KUKA KRL data list: $config.dat

&ACCESS RV
&PARAM DISKPATH = SYSTEM
&REL 3
DEFDAT $CONFIG
;FOLD BASISTECH GLOBALS
;==================================
; Default parameters for movement
; These values shouldn't be changed
;==================================

;----------------------------------
; general MOVEMENT - parameters:
;----------------------------------

INT DEF_OV_PRO=100
INT DEF_ADVANCE=3

; PTP - MOVEMENTS
;----------------------------------
INT DEF_VEL_PTP=100
INT DEF_ACC_PTP=50

; CP - MOVEMENTS
;----------------------------------
DECL CIRC_TYPE DEF_CIRC_TYP=#BASE
DECL JERK_STRUC DEF_JERK_STRUC={CP 500.0,ORI 50000.0,AX {A1 1000.0,A2 1000.0,A3 1000.0,A4 1000.0,A5 1000.0,A6 1000.0,E1 1000.0,E2 1000.0,E3 1000.0,E4 1000.0,E5 1000.0,E6 1000.0}}
REAL DEF_GEAR_JERK=100.0
REAL DEF_VEL_CP=2.0
REAL DEF_VEL_ORI1=200.0
REAL DEF_VEL_ORI2=200.0
REAL DEF_VEL_ORIS=200.0
REAL DEF_ACC_CP=2.3
REAL DEF_ACC_ORI1=100.0
REAL DEF_ACC_ORI2=100.0
REAL DEF_ACC_ORIS=200.0
REAL DEF_VEL_FACT=1.0
REAL DEF_ACC_SPTP=100.0

; APO - parameters
;--------------------------------
INT DEF_APO_CPTP=50
INT DEF_APO_CVEL=100
REAL DEF_APO_CDIS=3.0
REAL DEF_APO_CORI=5.0
REAL DEF_APO_CORIS=80.0

;==================================
; Structures:
;==================================
ENUM BAS_COMMAND INITMOV,ACC_CP,ACC_PTP,VEL_CP,VEL_PTP,ACC_GLUE,TOOL,BASE,EX_BASE,PTP_DAT,CP_DAT,OUT_SYNC,OUT_ASYNC,GROUP,FRAMES,PTP_PARAMS,CP_PARAMS
ENUM OUT_MODETYPE TRIGGER_,CONT_,STOP_
ENUM IPO_M_T NONE,TCP,BASE
ENUM APO_MODE_T CPTP,CDIS
STRUC DIG_OUT_TYPE INT FIRST_BIT, LENGTH, PARITY, CODING
STRUC CTRL_IN_T INT IN_NR, CHAR NAME_NAT[20]
STRUC CTRL_OUT_T INT OUT_NR, BOOL INI, CHAR NAME_NAT[20]
STRUC FCT_OUT_T INT NO, REAL PULS_TIME, BOOL STATE
STRUC FCT_IN_T INT NO, BOOL STATE
STRUC PDAT REAL VEL, ACC, APO_DIST, APO_MODE_T APO_MODE, REAL GEAR_JERK
STRUC LDAT REAL VEL, ACC, APO_DIST, APO_FAC, AXIS_VEL, AXIS_ACC, ORI_TYPE ORI_TYP, CIRC_TYPE CIRC_TYP, REAL JERK_FAC, GEAR_JERK, INT EXAX_IGN, CIRC_MODE CB
STRUC FDAT INT TOOL_NO, BASE_NO, IPO_MODE IPO_FRAME, CHAR POINT2[24], BOOL TQ_STATE
STRUC ODAT INT OUT_NO, BOOL STATE, REAL PULSE_TIME, OUT_MODETYPE OUT_MODE, REAL TIME_DELAY, OFFSET
STRUC BASIS_SUGG_T CHAR POINT1[24], POINT2[24], CP_PARAMS[24], PTP_PARAMS[24], CONT[24], CP_VEL[24], PTP_VEL[24], SYNC_PARAMS[24], SPL_NAME[24], A_PARAMS[24]

STRUC OUT_SUGG_T CHAR PARAMS[24]
STRUC MACHINE_DEF_T CHAR NAME[24], INT COOP_KRC_INDEX, CHAR PARENT[24], FRAME ROOT, ESYS MECH_TYPE, CHAR GEOMETRY[255]
STRUC MACHINE_TOOL_T INT MACH_DEF_INDEX, CHAR PARENT[24], CHAR GEOMETRY[255]
STRUC MACHINE_FRAME_T INT MACH_DEF_INDEX, CHAR PARENT[24], CHAR GEOMETRY[255]

STRUC TRIGGER_PARA INT TriggerPath, BOOL TriggerOnStart, INT TriggerDelay, CHAR TriggerTask[40]
STRUC CONSTVEL_PARA INT ConstVelTyp, INT ConstVelPath, BOOL ConstVelOnStart
STRUC CONDSTOP_PARA INT CondStopPath, BOOL CondStopOnStart, CHAR StopCondition[40]
STRUC ADAT TRIGGER_PARA TriggerPara, CONSTVEL_PARA ConstVelPara, CONDSTOP_PARA CondStopPara

;==================================
; TORQUE MONITORING
;==================================
SIGNAL sTQM_SPSACTIVE $IN[1026]
SIGNAL sTQM_SPSSTATUS $OUT[1024]

BOOL bTQM_ACTIVE=FALSE
BOOL bTQM_CYC=FALSE
BOOL bTQM_KCPSTATUS=TRUE

STRUC TM_SUGG_T CHAR TM_ID[24]
STRUC TQM_TQDAT_T INT T11, T12, T13, T14, T15, T16, T21, T22, T23, T24, T25, T26, K1, K2, K3, K4, K5, K6, O1, O2, ID, OVM, REAL TMF

DECL TQM_TQDAT_T TMDEFAULT={T11 200,T12 200,T13 200,T14 200,T15 200,T16 200,T21 1000,T22 1000,T23 1000,T24 1000,T25 1000,T26 1000,K1 280,K2 280,K3 280,K4 280,K5 280,K6 280,O1 20,O2 30,ID 0,OVM 0,TMF 1.0}
DECL TQM_TQDAT_T TM0={T11 200,T12 200,T13 200,T14 200,T15 200,T16 200,T21 1000,T22 1000,T23 1000,T24 1000,T25 1000,T26 1000,K1 280,K2 280,K3 280,K4 280,K5 280,K6 280,O1 20,O2 30,ID 0,OVM 0,TMF 1.0}

DECL TQM_TQDAT_T TQM_DATA_C[8]
DECL TQM_TQDAT_T TQM_TEMP

;==================================
; External declarations:
;==================================
EXT BAS (BAS_COMMAND :IN, REAL :IN )
EXT IR_STOPM ( )

;====================
; Signal declarations
; Do not change !!!!!
;====================
SIGNAL CHANNEL_1 $ANOUT[1]
SIGNAL CHANNEL_2 $ANOUT[2]
SIGNAL CHANNEL_3 $ANOUT[3]
SIGNAL CHANNEL_4 $ANOUT[4]
SIGNAL CHANNEL_5 $ANOUT[5]
SIGNAL CHANNEL_6 $ANOUT[6]
SIGNAL CHANNEL_7 $ANOUT[7]
SIGNAL CHANNEL_8 $ANOUT[8]
SIGNAL CHANNEL_9 $ANOUT[9]
SIGNAL CHANNEL_10 $ANOUT[10]
SIGNAL CHANNEL_11 $ANOUT[11]
SIGNAL CHANNEL_12 $ANOUT[12]
SIGNAL CHANNEL_13 $ANOUT[13]
SIGNAL CHANNEL_14 $ANOUT[14]
SIGNAL CHANNEL_15 $ANOUT[15]
SIGNAL CHANNEL_16 $ANOUT[16]
SIGNAL CHANNEL_17 $ANOUT[17]
SIGNAL CHANNEL_18 $ANOUT[18]
SIGNAL CHANNEL_19 $ANOUT[19]
SIGNAL CHANNEL_20 $ANOUT[20]
SIGNAL CHANNEL_21 $ANOUT[21]
SIGNAL CHANNEL_22 $ANOUT[22]
SIGNAL CHANNEL_23 $ANOUT[23]
SIGNAL CHANNEL_24 $ANOUT[24]
SIGNAL CHANNEL_25 $ANOUT[25]
SIGNAL CHANNEL_26 $ANOUT[26]
SIGNAL CHANNEL_27 $ANOUT[27]
SIGNAL CHANNEL_28 $ANOUT[28]
SIGNAL CHANNEL_29 $ANOUT[29]
SIGNAL CHANNEL_30 $ANOUT[30]
SIGNAL CHANNEL_31 $ANOUT[31]
SIGNAL CHANNEL_32 $ANOUT[32]

;==================================
; ID external user log-on:
;==================================
SIGNAL ExtUserID $IN[1026] TO $IN[1026]
SIGNAL ExtUserIDWatchDog $IN[1026]

;==================================
; Variables:
;==================================
DECL PDAT PDEFAULT={VEL 100.0,ACC 100.0,APO_DIST 100.0,GEAR_JERK 50.0}
DECL LDAT LDEFAULT={VEL 2.0,ACC 100.0,APO_DIST 100.0,APO_FAC 50.0,AXIS_VEL 100.0,AXIS_ACC 100.0,ORI_TYP #VAR,CIRC_TYP #BASE,JERK_FAC 50.0,GEAR_JERK 50.0,EXAX_IGN 0}
DECL LDAT CDEFAULT={CB {AUX_PT {ORI #CONSIDER,E1 #CONSIDER,E2 #CONSIDER,E3 #CONSIDER,E4 #CONSIDER,E5 #CONSIDER,E6 #CONSIDER},TARGET_PT {ORI #INTERPOLATE,E1 #INTERPOLATE,E2 #INTERPOLATE,E3 #INTERPOLATE,E4 #INTERPOLATE,E5 #INTERPOLATE,E6 #INTERPOLATE}}}
DECL FDAT FDEFAULT={TOOL_NO 1,BASE_NO 0,IPO_FRAME #BASE,POINT2[] " ",TQ_STATE FALSE}
DECL FDAT FHOME={TOOL_NO 1,BASE_NO 0,IPO_FRAME #BASE,POINT2[] " ",TQ_STATE FALSE}
DECL ODAT ODEFAULT={OUT_NO 1,STATE TRUE,PULSE_TIME 0.0,OUT_MODE #STOP_,TIME_DELAY 0.0,OFFSET 0.0}

DECL ADAT TDEFAULT={TriggerPara {TriggerPath 0,TriggerOnStart FALSE,TriggerDelay 0,TriggerTask[] " "}}
DECL ADAT CVDEFAULT={ConstVelPara {ConstVelTyp 0,ConstVelPath 0,ConstVelOnStart FALSE}}
DECL ADAT CSDEFAULT={CondStopPara {CondStopPath 0,CondStopOnStart FALSE,StopCondition[] " "}}

DECL PDAT PDAT_ACT
DECL LDAT LDAT_ACT
DECL FDAT FDAT_ACT
DECL ODAT ODAT_ACT
DECL INT ACT_FILTER
DECL INT ACT_DELAY
DECL INT ACT_DISTANCE

DECL CHAR SPL_NAME[24]

;GROUP-Definitions
;----------------------------------
INT COMPL_GROUP='B0001'

INT DEF_GROUP[10]
DEF_GROUP[1]='B1111'; complete
DEF_GROUP[2]='B0001'; robot only
DEF_GROUP[3]='B0011'; robot and track
DEF_GROUP[4]='B0111'; robot, track and ext. axis2
DEF_GROUP[5]='B1011'; robot, track and ext. axis3
DEF_GROUP[6]='B1111'; robot, track and ext. axis2+3
DEF_GROUP[7]='B1111'; complete
DEF_GROUP[8]='B1111'; complete
DEF_GROUP[9]='B1111'; complete
DEF_GROUP[10]='B1111'; complete

INT $ACT_GROUP='B0001'

; HOME POSITION
;----------------------------------
E6AXIS XHOME={A1 17.6205368,A2 -19.1096439,A3 94.6799545,A4 -1.38059322E-5,A5 14.4296818,A6 -163.685623,E1 0.0,E2 0.0,E3 0.0,E4 0.0,E5 0.0,E6 0.0}
E6AXIS XHOME1={A1 0.0,A2 -90.0,A3 90.0,A4 0.0,A5 0.0,A6 0.0,E1 0.0,E2 0.0,E3 0.0,E4 0.0,E5 0.0,E6 0.0}
E6AXIS XHOME2={A1 0.0,A2 -90.0,A3 90.0,A4 0.0,A5 0.0,A6 0.0,E1 0.0,E2 0.0,E3 0.0,E4 0.0,E5 0.0,E6 0.0}
E6AXIS XHOME3={A1 0.0,A2 -90.0,A3 90.0,A4 0.0,A5 0.0,A6 0.0,E1 0.0,E2 0.0,E3 0.0,E4 0.0,E5 0.0,E6 0.0}
E6AXIS XHOME4={A1 0.0,A2 -90.0,A3 90.0,A4 0.0,A5 0.0,A6 0.0,E1 0.0,E2 0.0,E3 0.0,E4 0.0,E5 0.0,E6 0.0}
E6AXIS XHOME5={A1 0.0,A2 -90.0,A3 90.0,A4 0.0,A5 0.0,A6 0.0,E1 0.0,E2 0.0,E3 0.0,E4 0.0,E5 0.0,E6 0.0}

; REFERENCE POINTS
;----------------------------------
DECL FRAME REF_PT[16]
REF_PT[1]={X 0.0,Y 0.0,Z 0.0,A 0.0,B 0.0,C 0.0}
REF_PT[2]={X 2325.62915,Y 305.171722,Z 689.508,A -0.650802493,B -2.90535426,C -176.880188}
REF_PT[3]={X 0.0,Y 0.0,Z 0.0,A 0.0,B 0.0,C 0.0}
REF_PT[4]={X 0.0,Y 0.0,Z 0.0,A 0.0,B 0.0,C 0.0}
REF_PT[5]={X 0.0,Y 0.0,Z 0.0,A 0.0,B 0.0,C 0.0}
REF_PT[6]={X 0.0,Y 0.0,Z 0.0,A 0.0,B 0.0,C 0.0}
REF_PT[7]={X 0.0,Y 0.0,Z 0.0,A 0.0,B 0.0,C 0.0}
REF_PT[8]={X 0.0,Y 0.0,Z 0.0,A 0.0,B 0.0,C 0.0}
REF_PT[9]={X 0.0,Y 0.0,Z 0.0,A 0.0,B 0.0,C 0.0}
REF_PT[10]={X 1725.46448,Y -99.6691,Z -810.829956,A -0.509644389,B -1.51949847,C 90.506424}
REF_PT[11]={X 0.0,Y 0.0,Z 0.0,A 0.0,B 0.0,C 0.0}
REF_PT[12]={X 0.0,Y 0.0,Z 0.0,A 0.0,B 0.0,C 0.0}
REF_PT[13]={X 0.0,Y 0.0,Z 0.0,A 0.0,B 0.0,C 0.0}
REF_PT[14]={X 0.0,Y 0.0,Z 0.0,A 0.0,B 0.0,C 0.0}
REF_PT[15]={X 0.0,Y 0.0,Z 0.0,A 0.0,B 0.0,C 0.0}
REF_PT[16]={X 0.0,Y 0.0,Z 0.0,A 0.0,B 0.0,C 0.0}

FRAME REF_TOOL={X 0.0,Y 0.0,Z 0.0,A 0.0,B 0.0,C 0.0}

; TOOL and BASE data
;----------------------------------
BOOL AUTO_IPO_M=FALSE
BOOL STOPM_FLAG=FALSE
BOOL TOOL_CORR_ON=FALSE
BOOL TOOL_CORR_W_ON=FALSE
BOOL BASE_CORR_ON=FALSE
BOOL M_BAS_COR_ON=FALSE
FRAME TOOL_CORR={X 0.0,Y 0.0,Z 0.0,A 0.0,B 0.0,C 0.0}
FRAME TOOL_CORR_W={X 0.0,Y 0.0,Z 0.0,A 0.0,B 0.0,C 0.0}
FRAME BASE_CORR={X 0.0,Y 0.0,Z 0.0,A 0.0,B 0.0,C 0.0}
FRAME M_BASE_CORR={X 0.0,Y 0.0,Z 0.0,A 0.0,B 0.0,C 0.0}
INT COR_TOOL_NO=0


INT MAX_TOOL=16
DECL FRAME TOOL_DATA[16]
TOOL_DATA[1]={X 0.0,Y 0.0,Z 600.0,A 0.0,B 0.0,C 0.0}
TOOL_DATA[2]={X 0.0,Y 0.0,Z 0.0,A 0.0,B 0.0,C 0.0}
TOOL_DATA[3]={X 0.0,Y 0.0,Z 0.0,A 0.0,B 0.0,C 0.0}
TOOL_DATA[4]={X 0.0,Y 0.0,Z 0.0,A 0.0,B 0.0,C 0.0}
TOOL_DATA[5]={X 0.0,Y 0.0,Z 0.0,A 0.0,B 0.0,C 0.0}
TOOL_DATA[6]={X 0.0,Y 0.0,Z 0.0,A 0.0,B 0.0,C 0.0}
TOOL_DATA[7]={X 0.0,Y 0.0,Z 0.0,A 0.0,B 0.0,C 0.0}
TOOL_DATA[8]={X 0.0,Y 0.0,Z 0.0,A 0.0,B 0.0,C 0.0}
TOOL_DATA[9]={X 0.0,Y 0.0,Z 0.0,A 0.0,B 0.0,C 0.0}
TOOL_DATA[10]={X 0.0,Y 0.0,Z 0.0,A 0.0,B 0.0,C 0.0}
TOOL_DATA[11]={X 0.0,Y 0.0,Z 0.0,A 0.0,B 0.0,C 0.0}
TOOL_DATA[12]={X 0.0,Y 0.0,Z 0.0,A 0.0,B 0.0,C 0.0}
TOOL_DATA[13]={X 0.0,Y 0.0,Z 0.0,A 0.0,B 0.0,C 0.0}
TOOL_DATA[14]={X 0.0,Y 0.0,Z 0.0,A 0.0,B 0.0,C 0.0}
TOOL_DATA[15]={X 0.0,Y 0.0,Z 0.0,A 0.0,B 0.0,C 0.0}
TOOL_DATA[16]={X 0.0,Y 0.0,Z 0.0,A 0.0,B 0.0,C 0.0}

DECL CHAR TOOL_NAME[16,24]
TOOL_NAME[1,]="GripperBP2"
TOOL_NAME[2,]=" "
TOOL_NAME[3,]=" "
TOOL_NAME[4,]=" "
TOOL_NAME[5,]=" "
TOOL_NAME[6,]=" "
TOOL_NAME[7,]=" "
TOOL_NAME[8,]=" "
TOOL_NAME[9,]=" "
TOOL_NAME[10,]=" "
TOOL_NAME[11,]=" "
TOOL_NAME[12,]=" "
TOOL_NAME[13,]=" "
TOOL_NAME[14,]=" "
TOOL_NAME[15,]=" "
TOOL_NAME[16,]=" "

DECL LOAD LOAD_DATA[16]
LOAD_DATA[1]={M 100.0,CM {X 0.0,Y 0.0,Z -0.38,A 0.0,B 0.0,C 0.0},J {X 32.66,Y 31.81,Z 15.25}}
LOAD_DATA[2]={M -1.0,CM {X 0.0,Y 0.0,Z 0.0,A 0.0,B 0.0,C 0.0},J {X 0.0,Y 0.0,Z 0.0}}
LOAD_DATA[3]={M -1.0,CM {X 0.0,Y 0.0,Z 0.0,A 0.0,B 0.0,C 0.0},J {X 0.0,Y 0.0,Z 0.0}}
LOAD_DATA[4]={M -1.0,CM {X 0.0,Y 0.0,Z 0.0,A 0.0,B 0.0,C 0.0},J {X 0.0,Y 0.0,Z 0.0}}
LOAD_DATA[5]={M -1.0,CM {X 0.0,Y 0.0,Z 0.0,A 0.0,B 0.0,C 0.0},J {X 0.0,Y 0.0,Z 0.0}}
LOAD_DATA[6]={M -1.0,CM {X 0.0,Y 0.0,Z 0.0,A 0.0,B 0.0,C 0.0},J {X 0.0,Y 0.0,Z 0.0}}
LOAD_DATA[7]={M -1.0,CM {X 0.0,Y 0.0,Z 0.0,A 0.0,B 0.0,C 0.0},J {X 0.0,Y 0.0,Z 0.0}}
LOAD_DATA[8]={M -1.0,CM {X 0.0,Y 0.0,Z 0.0,A 0.0,B 0.0,C 0.0},J {X 0.0,Y 0.0,Z 0.0}}
LOAD_DATA[9]={M -1.0,CM {X 0.0,Y 0.0,Z 0.0,A 0.0,B 0.0,C 0.0},J {X 0.0,Y 0.0,Z 0.0}}
LOAD_DATA[10]={M -1.0,CM {X 0.0,Y 0.0,Z 0.0,A 0.0,B 0.0,C 0.0},J {X 0.0,Y 0.0,Z 0.0}}
LOAD_DATA[11]={M -1.0,CM {X 0.0,Y 0.0,Z 0.0,A 0.0,B 0.0,C 0.0},J {X 0.0,Y 0.0,Z 0.0}}
LOAD_DATA[12]={M -1.0,CM {X 0.0,Y 0.0,Z 0.0,A 0.0,B 0.0,C 0.0},J {X 0.0,Y 0.0,Z 0.0}}
LOAD_DATA[13]={M -1.0,CM {X 0.0,Y 0.0,Z 0.0,A 0.0,B 0.0,C 0.0},J {X 0.0,Y 0.0,Z 0.0}}
LOAD_DATA[14]={M -1.0,CM {X 0.0,Y 0.0,Z 0.0,A 0.0,B 0.0,C 0.0},J {X 0.0,Y 0.0,Z 0.0}}
LOAD_DATA[15]={M -1.0,CM {X 0.0,Y 0.0,Z 0.0,A 0.0,B 0.0,C 0.0},J {X 0.0,Y 0.0,Z 0.0}}
LOAD_DATA[16]={M -1.0,CM {X 0.0,Y 0.0,Z 0.0,A 0.0,B 0.0,C 0.0},J {X 0.0,Y 0.0,Z 0.0}}

DECL IPO_M_T TOOL_TYPE[16]
TOOL_TYPE[1]=#BASE
TOOL_TYPE[2]=#NONE
TOOL_TYPE[3]=#NONE
TOOL_TYPE[4]=#NONE
TOOL_TYPE[5]=#NONE
TOOL_TYPE[6]=#NONE
TOOL_TYPE[7]=#NONE
TOOL_TYPE[8]=#NONE
TOOL_TYPE[9]=#NONE
TOOL_TYPE[10]=#NONE
TOOL_TYPE[11]=#NONE
TOOL_TYPE[12]=#NONE
TOOL_TYPE[13]=#NONE
TOOL_TYPE[14]=#NONE
TOOL_TYPE[15]=#NONE
TOOL_TYPE[16]=#NONE

DECL LOAD LOAD_A1_DATA={M -1.0,CM {X 0.0,Y 0.0,Z 0.0,A 0.0,B 0.0,C 0.0},J {X 0.0,Y 0.0,Z 0.0}}
DECL LOAD LOAD_A2_DATA={M -1.0,CM {X 0.0,Y 0.0,Z 0.0,A 0.0,B 0.0,C 0.0},J {X 0.0,Y 0.0,Z 0.0}}
DECL LOAD LOAD_A3_DATA={M -1.0,CM {X 0.0,Y 0.0,Z 0.0,A 0.0,B 0.0,C 0.0},J {X 0.0,Y 0.0,Z 0.0}}


INT MAX_BASE=32
DECL FRAME BASE_DATA[32]
BASE_DATA[1]={X -870.0,Y 580.0,Z -600.0,A 28.0,B 0.0,C 0.0}
BASE_DATA[2]={X -1070.0,Y -2850.0,Z -1150.0,A -1.2,B 0.0,C 0.0}
BASE_DATA[3]={X 1811.80701,Y 1245.51,Z -697.576172,A 44.1548,B 0.0,C 0.0}
BASE_DATA[4]={X 302.249908,Y 1595.83398,Z -599.960693,A -39.6942,B 0.0,C 0.0}
BASE_DATA[5]={X -852.160828,Y -2828.22412,Z -599.959717,A 0.0,B 0.0,C 0.0}
BASE_DATA[6]={X 0.0,Y 0.0,Z 0.0,A 0.0,B 0.0,C 0.0}
BASE_DATA[7]={X 0.0,Y 0.0,Z 0.0,A 0.0,B 0.0,C 0.0}
BASE_DATA[8]={X 0.0,Y 0.0,Z 0.0,A 0.0,B 0.0,C 0.0}
BASE_DATA[9]={X 0.0,Y 0.0,Z 0.0,A 0.0,B 0.0,C 0.0}
BASE_DATA[10]={X 0.0,Y 0.0,Z 0.0,A 0.0,B 0.0,C 0.0}
BASE_DATA[11]={X 0.0,Y 0.0,Z 0.0,A 0.0,B 0.0,C 0.0}
BASE_DATA[12]={X 0.0,Y 0.0,Z 0.0,A 0.0,B 0.0,C 0.0}
BASE_DATA[13]={X 0.0,Y 0.0,Z 0.0,A 0.0,B 0.0,C 0.0}
BASE_DATA[14]={X 0.0,Y 0.0,Z 0.0,A 0.0,B 0.0,C 0.0}
BASE_DATA[15]={X 0.0,Y 0.0,Z 0.0,A 0.0,B 0.0,C 0.0}
BASE_DATA[16]={X 0.0,Y 0.0,Z 0.0,A 0.0,B 0.0,C 0.0}
BASE_DATA[17]={X 0.0,Y 0.0,Z 0.0,A 0.0,B 0.0,C 0.0}
BASE_DATA[18]={X 0.0,Y 0.0,Z 0.0,A 0.0,B 0.0,C 0.0}
BASE_DATA[19]={X 0.0,Y 0.0,Z 0.0,A 0.0,B 0.0,C 0.0}
BASE_DATA[20]={X 0.0,Y 0.0,Z 0.0,A 0.0,B 0.0,C 0.0}
BASE_DATA[21]={X 0.0,Y 0.0,Z 0.0,A 0.0,B 0.0,C 0.0}
BASE_DATA[22]={X 0.0,Y 0.0,Z 0.0,A 0.0,B 0.0,C 0.0}
BASE_DATA[23]={X 0.0,Y 0.0,Z 0.0,A 0.0,B 0.0,C 0.0}
BASE_DATA[24]={X 0.0,Y 0.0,Z 0.0,A 0.0,B 0.0,C 0.0}
BASE_DATA[25]={X 0.0,Y 0.0,Z 0.0,A 0.0,B 0.0,C 0.0}
BASE_DATA[26]={X 0.0,Y 0.0,Z 0.0,A 0.0,B 0.0,C 0.0}
BASE_DATA[27]={X 0.0,Y 0.0,Z 0.0,A 0.0,B 0.0,C 0.0}
BASE_DATA[28]={X 0.0,Y 0.0,Z 0.0,A 0.0,B 0.0,C 0.0}
BASE_DATA[29]={X 0.0,Y 0.0,Z 0.0,A 0.0,B 0.0,C 0.0}
BASE_DATA[30]={X 0.0,Y 0.0,Z 0.0,A 0.0,B 0.0,C 0.0}
BASE_DATA[31]={X 0.0,Y 0.0,Z 0.0,A 0.0,B 0.0,C 0.0}
BASE_DATA[32]={X 0.0,Y 0.0,Z 0.0,A 0.0,B 0.0,C 0.0}

DECL CHAR BASE_NAME[32,24]
BASE_NAME[1,]="PalletLeft"
BASE_NAME[2,]="PalletRight"
BASE_NAME[3,]="PikupBase"
BASE_NAME[4,]="10kgLftBas"
BASE_NAME[5,]="10kgRghBas"
BASE_NAME[6,]=" "
BASE_NAME[7,]=" "
BASE_NAME[8,]=" "
BASE_NAME[9,]=" "
BASE_NAME[10,]="KukaReburn"
BASE_NAME[11,]=" "
BASE_NAME[12,]=" "
BASE_NAME[13,]=" "
BASE_NAME[14,]=" "
BASE_NAME[15,]=" "
BASE_NAME[16,]=" "
BASE_NAME[17,]=" "
BASE_NAME[18,]=" "
BASE_NAME[19,]=" "
BASE_NAME[20,]=" "
BASE_NAME[21,]=" "
BASE_NAME[22,]=" "
BASE_NAME[23,]=" "
BASE_NAME[24,]=" "
BASE_NAME[25,]=" "
BASE_NAME[26,]=" "
BASE_NAME[27,]=" "
BASE_NAME[28,]=" "
BASE_NAME[29,]=" "
BASE_NAME[30,]=" "
BASE_NAME[31,]=" "
BASE_NAME[32,]=" "


DECL IPO_M_T BASE_TYPE[32]
BASE_TYPE[1]=#BASE
BASE_TYPE[2]=#BASE
BASE_TYPE[3]=#BASE
BASE_TYPE[4]=#BASE
BASE_TYPE[5]=#BASE
BASE_TYPE[6]=#NONE
BASE_TYPE[7]=#NONE
BASE_TYPE[8]=#NONE
BASE_TYPE[9]=#NONE
BASE_TYPE[10]=#NONE
BASE_TYPE[11]=#NONE
BASE_TYPE[12]=#NONE
BASE_TYPE[13]=#NONE
BASE_TYPE[14]=#NONE
BASE_TYPE[15]=#NONE
BASE_TYPE[16]=#NONE
BASE_TYPE[17]=#NONE
BASE_TYPE[18]=#NONE
BASE_TYPE[19]=#NONE
BASE_TYPE[20]=#NONE
BASE_TYPE[21]=#NONE
BASE_TYPE[22]=#NONE
BASE_TYPE[23]=#NONE
BASE_TYPE[24]=#NONE
BASE_TYPE[25]=#NONE
BASE_TYPE[26]=#NONE
BASE_TYPE[27]=#NONE
BASE_TYPE[28]=#NONE
BASE_TYPE[29]=#NONE
BASE_TYPE[30]=#NONE
BASE_TYPE[31]=#NONE
BASE_TYPE[32]=#NONE

;******************************************
; Variables for CELL DEFINITION
;******************************************

INT MAX_MACHINES=16
DECL MACHINE_DEF_T MACHINE_DEF[16]
MACHINE_DEF[1]={NAME[] "KR 210 R3300 K ultra",COOP_KRC_INDEX 1,PARENT[] "WORLD",ROOT {X 0.0,Y 0.0,Z 0.0,A 0.0,B 0.0,C 0.0},MECH_TYPE #ROBOT,GEOMETRY[] "ObjectId = 536625629"}
MACHINE_DEF[2]={NAME[] " ",COOP_KRC_INDEX 0,PARENT[] " ",ROOT {X 0.0,Y 0.0,Z 0.0,A 0.0,B 0.0,C 0.0},MECH_TYPE #NONE,GEOMETRY[] " "}
MACHINE_DEF[3]={NAME[] " ",COOP_KRC_INDEX 0,PARENT[] " ",ROOT {X 0.0,Y 0.0,Z 0.0,A 0.0,B 0.0,C 0.0},MECH_TYPE #NONE,GEOMETRY[] " "}
MACHINE_DEF[4]={NAME[] " ",COOP_KRC_INDEX 0,PARENT[] " ",ROOT {X 0.0,Y 0.0,Z 0.0,A 0.0,B 0.0,C 0.0},MECH_TYPE #NONE,GEOMETRY[] " "}
MACHINE_DEF[5]={NAME[] " ",COOP_KRC_INDEX 0,PARENT[] " ",ROOT {X 0.0,Y 0.0,Z 0.0,A 0.0,B 0.0,C 0.0},MECH_TYPE #NONE,GEOMETRY[] " "}
MACHINE_DEF[6]={NAME[] " ",COOP_KRC_INDEX 0,PARENT[] " ",ROOT {X 0.0,Y 0.0,Z 0.0,A 0.0,B 0.0,C 0.0},MECH_TYPE #NONE,GEOMETRY[] " "}
MACHINE_DEF[7]={NAME[] " ",COOP_KRC_INDEX 0,PARENT[] " ",ROOT {X 0.0,Y 0.0,Z 0.0,A 0.0,B 0.0,C 0.0},MECH_TYPE #NONE,GEOMETRY[] " "}
MACHINE_DEF[8]={NAME[] " ",COOP_KRC_INDEX 0,PARENT[] " ",ROOT {X 0.0,Y 0.0,Z 0.0,A 0.0,B 0.0,C 0.0},MECH_TYPE #NONE,GEOMETRY[] " "}
MACHINE_DEF[9]={NAME[] " ",COOP_KRC_INDEX 0,PARENT[] " ",ROOT {X 0.0,Y 0.0,Z 0.0,A 0.0,B 0.0,C 0.0},MECH_TYPE #NONE,GEOMETRY[] " "}
MACHINE_DEF[10]={NAME[] " ",COOP_KRC_INDEX 0,PARENT[] " ",ROOT {X 0.0,Y 0.0,Z 0.0,A 0.0,B 0.0,C 0.0},MECH_TYPE #NONE,GEOMETRY[] " "}
MACHINE_DEF[11]={NAME[] " ",COOP_KRC_INDEX 0,PARENT[] " ",ROOT {X 0.0,Y 0.0,Z 0.0,A 0.0,B 0.0,C 0.0},MECH_TYPE #NONE,GEOMETRY[] " "}
MACHINE_DEF[12]={NAME[] " ",COOP_KRC_INDEX 0,PARENT[] " ",ROOT {X 0.0,Y 0.0,Z 0.0,A 0.0,B 0.0,C 0.0},MECH_TYPE #NONE,GEOMETRY[] " "}
MACHINE_DEF[13]={NAME[] " ",COOP_KRC_INDEX 0,PARENT[] " ",ROOT {X 0.0,Y 0.0,Z 0.0,A 0.0,B 0.0,C 0.0},MECH_TYPE #NONE,GEOMETRY[] " "}
MACHINE_DEF[14]={NAME[] " ",COOP_KRC_INDEX 0,PARENT[] " ",ROOT {X 0.0,Y 0.0,Z 0.0,A 0.0,B 0.0,C 0.0},MECH_TYPE #NONE,GEOMETRY[] " "}
MACHINE_DEF[15]={NAME[] " ",COOP_KRC_INDEX 0,PARENT[] " ",ROOT {X 0.0,Y 0.0,Z 0.0,A 0.0,B 0.0,C 0.0},MECH_TYPE #NONE,GEOMETRY[] " "}
MACHINE_DEF[16]={NAME[] " ",COOP_KRC_INDEX 0,PARENT[] " ",ROOT {X 0.0,Y 0.0,Z 0.0,A 0.0,B 0.0,C 0.0},MECH_TYPE #NONE,GEOMETRY[] " "}

DECL MACHINE_TOOL_T MACHINE_TOOL_DAT[16]
MACHINE_TOOL_DAT[1]={MACH_DEF_INDEX 1,PARENT[] "KR 210 R3300 K ultra",GEOMETRY[] " "}
MACHINE_TOOL_DAT[2]={MACH_DEF_INDEX 0,PARENT[] " ",GEOMETRY[] " "}
MACHINE_TOOL_DAT[3]={MACH_DEF_INDEX 0,PARENT[] " ",GEOMETRY[] " "}
MACHINE_TOOL_DAT[4]={MACH_DEF_INDEX 0,PARENT[] " ",GEOMETRY[] " "}
MACHINE_TOOL_DAT[5]={MACH_DEF_INDEX 0,PARENT[] " ",GEOMETRY[] " "}
MACHINE_TOOL_DAT[6]={MACH_DEF_INDEX 0,PARENT[] " ",GEOMETRY[] " "}
MACHINE_TOOL_DAT[7]={MACH_DEF_INDEX 0,PARENT[] " ",GEOMETRY[] " "}
MACHINE_TOOL_DAT[8]={MACH_DEF_INDEX 0,PARENT[] " ",GEOMETRY[] " "}
MACHINE_TOOL_DAT[9]={MACH_DEF_INDEX 0,PARENT[] " ",GEOMETRY[] " "}
MACHINE_TOOL_DAT[10]={MACH_DEF_INDEX 0,PARENT[] " ",GEOMETRY[] " "}
MACHINE_TOOL_DAT[11]={MACH_DEF_INDEX 0,PARENT[] " ",GEOMETRY[] " "}
MACHINE_TOOL_DAT[12]={MACH_DEF_INDEX 0,PARENT[] " ",GEOMETRY[] " "}
MACHINE_TOOL_DAT[13]={MACH_DEF_INDEX 0,PARENT[] " ",GEOMETRY[] " "}
MACHINE_TOOL_DAT[14]={MACH_DEF_INDEX 0,PARENT[] " ",GEOMETRY[] " "}
MACHINE_TOOL_DAT[15]={MACH_DEF_INDEX 0,PARENT[] " ",GEOMETRY[] " "}
MACHINE_TOOL_DAT[16]={MACH_DEF_INDEX 0,PARENT[] " ",GEOMETRY[] " "}

DECL MACHINE_FRAME_T MACHINE_FRAME_DAT[32]
MACHINE_FRAME_DAT[1]={MACH_DEF_INDEX 0,PARENT[] "WORLD",GEOMETRY[] " "}
MACHINE_FRAME_DAT[2]={MACH_DEF_INDEX 0,PARENT[] "WORLD",GEOMETRY[] " "}
MACHINE_FRAME_DAT[3]={MACH_DEF_INDEX 0,PARENT[] "WORLD",GEOMETRY[] " "}
MACHINE_FRAME_DAT[4]={MACH_DEF_INDEX 0,PARENT[] "WORLD",GEOMETRY[] " "}
MACHINE_FRAME_DAT[5]={MACH_DEF_INDEX 0,PARENT[] "WORLD",GEOMETRY[] " "}
MACHINE_FRAME_DAT[6]={MACH_DEF_INDEX 0,PARENT[] " ",GEOMETRY[] " "}
MACHINE_FRAME_DAT[7]={MACH_DEF_INDEX 0,PARENT[] " ",GEOMETRY[] " "}
MACHINE_FRAME_DAT[8]={MACH_DEF_INDEX 0,PARENT[] " ",GEOMETRY[] " "}
MACHINE_FRAME_DAT[9]={MACH_DEF_INDEX 0,PARENT[] " ",GEOMETRY[] " "}
MACHINE_FRAME_DAT[10]={MACH_DEF_INDEX 0,PARENT[] " ",GEOMETRY[] " "}
MACHINE_FRAME_DAT[11]={MACH_DEF_INDEX 0,PARENT[] " ",GEOMETRY[] " "}
MACHINE_FRAME_DAT[12]={MACH_DEF_INDEX 0,PARENT[] " ",GEOMETRY[] " "}
MACHINE_FRAME_DAT[13]={MACH_DEF_INDEX 0,PARENT[] " ",GEOMETRY[] " "}
MACHINE_FRAME_DAT[14]={MACH_DEF_INDEX 0,PARENT[] " ",GEOMETRY[] " "}
MACHINE_FRAME_DAT[15]={MACH_DEF_INDEX 0,PARENT[] " ",GEOMETRY[] " "}
MACHINE_FRAME_DAT[16]={MACH_DEF_INDEX 0,PARENT[] " ",GEOMETRY[] " "}
MACHINE_FRAME_DAT[17]={MACH_DEF_INDEX 0,PARENT[] " ",GEOMETRY[] " "}
MACHINE_FRAME_DAT[18]={MACH_DEF_INDEX 0,PARENT[] " ",GEOMETRY[] " "}
MACHINE_FRAME_DAT[19]={MACH_DEF_INDEX 0,PARENT[] " ",GEOMETRY[] " "}
MACHINE_FRAME_DAT[20]={MACH_DEF_INDEX 0,PARENT[] " ",GEOMETRY[] " "}
MACHINE_FRAME_DAT[21]={MACH_DEF_INDEX 0,PARENT[] " ",GEOMETRY[] " "}
MACHINE_FRAME_DAT[22]={MACH_DEF_INDEX 0,PARENT[] " ",GEOMETRY[] " "}
MACHINE_FRAME_DAT[23]={MACH_DEF_INDEX 0,PARENT[] " ",GEOMETRY[] " "}
MACHINE_FRAME_DAT[24]={MACH_DEF_INDEX 0,PARENT[] " ",GEOMETRY[] " "}
MACHINE_FRAME_DAT[25]={MACH_DEF_INDEX 0,PARENT[] " ",GEOMETRY[] " "}
MACHINE_FRAME_DAT[26]={MACH_DEF_INDEX 0,PARENT[] " ",GEOMETRY[] " "}
MACHINE_FRAME_DAT[27]={MACH_DEF_INDEX 0,PARENT[] " ",GEOMETRY[] " "}
MACHINE_FRAME_DAT[28]={MACH_DEF_INDEX 0,PARENT[] " ",GEOMETRY[] " "}
MACHINE_FRAME_DAT[29]={MACH_DEF_INDEX 0,PARENT[] " ",GEOMETRY[] " "}
MACHINE_FRAME_DAT[30]={MACH_DEF_INDEX 0,PARENT[] " ",GEOMETRY[] " "}
MACHINE_FRAME_DAT[31]={MACH_DEF_INDEX 0,PARENT[] " ",GEOMETRY[] " "}
MACHINE_FRAME_DAT[32]={MACH_DEF_INDEX 0,PARENT[] " ",GEOMETRY[] " "}

;******************************************
; Variables for axis CALIBRATING
;******************************************
DECL INT CAL_AXIS
BOOL CONST_SPEED

;******************************************
; Variables for added TechPackages
;******************************************
INT POWER

;******************************************
; General purpose return value of functions
; like INVERSE, FORWARD
;******************************************
INT ERR_STATUS=-1

;******************************************
; Variables for TOUCHUP user limit
;******************************************
BOOL UM_TOUCHUP=FALSE
REAL CARTESIAN_TOL=5.0
REAL ROTATION_ANGLE=10.0
REAL EXTAX_TOL[6]
EXTAX_TOL[1]=10.0
EXTAX_TOL[2]=10.0
EXTAX_TOL[3]=10.0
EXTAX_TOL[4]=10.0
EXTAX_TOL[5]=10.0
EXTAX_TOL[6]=10.0

;******************************************
; Variables for Displaying and Konfiguring
;******************************************
DECL INT I[20]

I[1]=0
I[2]=0
I[3]=0
I[4]=0
I[5]=0
I[6]=0
I[7]=0
I[8]=0
I[9]=0
I[10]=0
I[11]=0
I[12]=0
I[13]=0
I[14]=0
I[15]=0
I[16]=0
I[17]=0
I[18]=0
I[19]=0
I[20]=0

;******************************************
; all for InterBus Mapping on optional segments
;******************************************

DECL INT IBUS_SEGMENT[16]
IBUS_SEGMENT[1]=0
IBUS_SEGMENT[2]=0
IBUS_SEGMENT[3]=0
IBUS_SEGMENT[4]=0
IBUS_SEGMENT[5]=0
IBUS_SEGMENT[6]=0
IBUS_SEGMENT[7]=0
IBUS_SEGMENT[8]=0
IBUS_SEGMENT[9]=0
IBUS_SEGMENT[10]=0
IBUS_SEGMENT[11]=0
IBUS_SEGMENT[12]=0
IBUS_SEGMENT[13]=0
IBUS_SEGMENT[14]=0
IBUS_SEGMENT[15]=0
IBUS_SEGMENT[16]=0

;******************************************
; Reduction factors
;******************************************
DECL REAL RedVelExAx[6]
RedVelExAx[1]=100.0
RedVelExAx[2]=100.0
RedVelExAx[3]=100.0
RedVelExAx[4]=100.0
RedVelExAx[5]=100.0
RedVelExAx[6]=100.0
DECL REAL RedAccExAx[6]
RedAccExAx[1]=100.0
RedAccExAx[2]=100.0
RedAccExAx[3]=100.0
RedAccExAx[4]=100.0
RedAccExAx[5]=100.0
RedAccExAx[6]=100.0
;ENDFOLD (BASISTECH GLOBALS)
;FOLD AUTOEXT GLOBALS
;==================================
; Structures:
;==================================
ENUM FUNCT_TYPE PGNO_GET,PGNO_ACKN,PGNO_FAULT
ENUM P00_COMMAND INIT_EXT,EXT_PGNO,CHK_HOME,EXT_ERR

STRUC SPS_PROG_TYPE INT PROG_NR, CHAR PROG_NAME[12]
;==================================
; External declarations:
;==================================
EXT P00 (P00_COMMAND :IN, FUNCT_TYPE :IN, CHAR[] :OUT, INT :IN )
;External declaration  for  Submit controlled AutoExt
EXT P00_SUBM (P00_COMMAND :IN, FUNCT_TYPE :IN )

;==================================
; Variables:
;==================================
; Variables for internal
; Communication:
;----------------------------------
BOOL ERROR_FLAG
BOOL CHECK_HOME=TRUE
BOOL PROG_CONTROL=FALSE
DECL CHAR PRO_NAME1_L[8]
PRO_NAME1_L[]="        "
DECL CHAR PRO_NAME1_A[8]
PRO_NAME1_A[]="        "

INT PGNO=0;copy of ext. pgno
INT PGNO_ERROR=0;transmission error
INT PGNO_TYPE=1;coding type of ext. pgno
INT REFLECT_PROG_NR=0; enable mirroring of program number inputs (1=enabled, 0=disabled)

; Variables for External
; Communication: I/O-Interface
;----------------------------------
INT PGNO_FBIT=33;first bit of ext. pgno input $IN[]
INT PGNO_FBIT_REFL=999;first bit of ext. pgno reflection output $OUT[]
INT PGNO_LENGTH=8;length of ext. pgno (max. 16)
INT PGNO_PARITY=41;parity bit of ext. pgno
INT PGNO_REQ=41;request ext. pgno input
INT PGNO_VALID=42;validate ext. pgno input
INT APPL_RUN=40;application program is running output
INT ERR_TO_PLC=35;error output to PLC
INT P01_STEP
INT CHK_STEP
INT PGNO_FLAG

; Table for assign SPS program number to program name
INT MAX_SPS_PROG=12
DECL SPS_PROG_TYPE SPS_PROG[12]
SPS_PROG[1]={PROG_NR 1,PROG_NAME[] "HP01()    "}
SPS_PROG[2]={PROG_NR 2,PROG_NAME[] "HP02()    "}
SPS_PROG[3]={PROG_NR 3,PROG_NAME[] "HP03()    "}
SPS_PROG[4]={PROG_NR 4,PROG_NAME[] "HP04()    "}
SPS_PROG[5]={PROG_NR 5,PROG_NAME[] "HP05()    "}
SPS_PROG[6]={PROG_NR 6,PROG_NAME[] "HP06()    "}
SPS_PROG[7]={PROG_NR 7,PROG_NAME[] "HP07()    "}
SPS_PROG[8]={PROG_NR 8,PROG_NAME[] "HP08()    "}
SPS_PROG[9]={PROG_NR 9,PROG_NAME[] "HP09()    "}
SPS_PROG[10]={PROG_NR 10,PROG_NAME[] "HP10()    "}
SPS_PROG[11]={PROG_NR 62,PROG_NAME[] "HP62()    "}
SPS_PROG[12]={PROG_NR 63,PROG_NAME[] "HP63()    "}
DECL CHAR TMPNAME[128]
TMPNAME[]="                                "
;ENDFOLD (AUTOEXT GLOBALS)
;FOLD BackupManagerConfig
BOOL BM_ENABLED
INT BM_OUTPUTVALUE
SIGNAL BM_OutputSignal $OUT[4095] TO $OUT[4096]
SIGNAL BM_InputSignal $IN[1026] TO $IN[1026]
;ENDFOLD BackupManagerConfig
;FOLD Conveyor
DECL INT CONV_PART_NBR[16]
CONV_PART_NBR[1]=0
CONV_PART_NBR[2]=0
CONV_PART_NBR[3]=0
CONV_PART_NBR[4]=0
CONV_PART_NBR[5]=0
CONV_PART_NBR[6]=0
CONV_PART_NBR[7]=0
CONV_PART_NBR[8]=0
CONV_PART_NBR[9]=0
CONV_PART_NBR[10]=0
CONV_PART_NBR[11]=0
CONV_PART_NBR[12]=0
CONV_PART_NBR[13]=0
CONV_PART_NBR[14]=0
CONV_PART_NBR[15]=0
CONV_PART_NBR[16]=0
;ENDFOLD Conveyor
;FOLD GRIPPERTECH GLOBALS
;==================================
; Structures:
;==================================
ENUM ON_OFF_TYP ON,OFF,MID
ENUM APO_TYP YES,NO
ENUM COMMAND OPN,CLO

STRUC GRP_TYP APO_TYP G_APO, REAL GRP_TIME, ON_OFF_TYP CTRL, INT DLY, INT DST
; structure for gripper definition
STRUC GRP_TYPES INT TYPE, OUT1, OUT2, OUT3, OUT4, IN1, IN2, IN3, IN4, GRP_OLD
; structure for last values
STRUC GRP_SUGG_T CHAR NUMBER[24], STATE[24], PARAMS[24]

;==================================
; External declarations:
;==================================
EXT H50 (INT :IN, INT :IN, INT :IN, GRP_TYP :IN )
EXT USER_GRP (INT :IN, INT :IN, INT :IN, GRP_TYP :IN )
;==================================
; Variables:
;==================================
; instruction codes
INT GRP=1
INT CHK_APO=2
INT GRP_APO=3
INT CHK_APO_UP=4
INT ZANGEN_FUNKT=0
INT AKT_ZANGE=1

;==================================
; Variables:
;==================================
DECL GRP_TYP GDEFAULT={G_APO #NO,GRP_TIME 0.2,CTRL #OFF,DLY 0,DST 1}
INT DUMMY=0

;constant for time out in sec
REAL TIME_OUT=3.0
INT CHK_CODE=0
BOOL APO_CHK_ON=FALSE
BOOL H50_FERTIG=FALSE

;==================================
; Options:
;==================================
BOOL APO_CHK_OPT=TRUE

;==================================
; Definition of grippers
;==================================
INT MAXGRIPPER=16

DECL GRP_TYPES GRIPPER[16]

GRIPPER[1]={TYPE 0,OUT1 1,OUT2 999,OUT3 999,OUT4 999,IN1 0,IN2 0,IN3 0,IN4 0,GRP_OLD 1}
GRIPPER[2]={TYPE 0,OUT1 2,OUT2 999,OUT3 999,OUT4 999,IN1 0,IN2 0,IN3 0,IN4 0,GRP_OLD 1}
GRIPPER[3]={TYPE 0,OUT1 3,OUT2 999,OUT3 999,OUT4 999,IN1 0,IN2 0,IN3 0,IN4 0,GRP_OLD 1}
GRIPPER[4]={TYPE 0,OUT1 999,OUT2 999,OUT3 999,OUT4 999,IN1 0,IN2 0,IN3 0,IN4 0,GRP_OLD 1}
GRIPPER[5]={TYPE 0,OUT1 999,OUT2 999,OUT3 999,OUT4 999,IN1 0,IN2 0,IN3 0,IN4 0,GRP_OLD 1}
GRIPPER[6]={TYPE 0,OUT1 999,OUT2 999,OUT3 999,OUT4 999,IN1 0,IN2 0,IN3 0,IN4 0,GRP_OLD 1}
GRIPPER[7]={TYPE 0,OUT1 999,OUT2 999,OUT3 999,OUT4 999,IN1 0,IN2 0,IN3 0,IN4 0,GRP_OLD 1}
GRIPPER[8]={TYPE 0,OUT1 999,OUT2 999,OUT3 999,OUT4 999,IN1 0,IN2 0,IN3 0,IN4 0,GRP_OLD 1}
GRIPPER[9]={TYPE 0,OUT1 999,OUT2 999,OUT3 999,OUT4 999,IN1 0,IN2 0,IN3 0,IN4 0,GRP_OLD 1}
GRIPPER[10]={TYPE 0,OUT1 999,OUT2 999,OUT3 999,OUT4 999,IN1 0,IN2 0,IN3 0,IN4 0,GRP_OLD 1}
GRIPPER[11]={TYPE 0,OUT1 999,OUT2 999,OUT3 999,OUT4 999,IN1 0,IN2 0,IN3 0,IN4 0,GRP_OLD 1}
GRIPPER[12]={TYPE 0,OUT1 999,OUT2 999,OUT3 999,OUT4 999,IN1 0,IN2 0,IN3 0,IN4 0,GRP_OLD 1}
GRIPPER[13]={TYPE 0,OUT1 999,OUT2 999,OUT3 999,OUT4 999,IN1 0,IN2 0,IN3 0,IN4 0,GRP_OLD 1}
GRIPPER[14]={TYPE 0,OUT1 999,OUT2 999,OUT3 999,OUT4 999,IN1 0,IN2 0,IN3 0,IN4 0,GRP_OLD 1}
GRIPPER[15]={TYPE 0,OUT1 999,OUT2 999,OUT3 999,OUT4 999,IN1 0,IN2 0,IN3 0,IN4 0,GRP_OLD 1}
GRIPPER[16]={TYPE 0,OUT1 999,OUT2 999,OUT3 999,OUT4 999,IN1 0,IN2 0,IN3 0,IN4 0,GRP_OLD 1}

REAL GRP_PULSE_TI=0.5; pulse time for gripper type 5
;ENDFOLD (GRIPPERTECH GLOBALS)
;FOLD SPOTTECH GLOBALS
;==================================
; Structures:
;==================================
ENUM S_COMMAND SPOT,RETR,PRESPOT,INIT,ADVSPOT
ENUM S_PAIR_SLCT FIRST,SECOND,BOTH

STRUC SPOT_SUGG_T CHAR GUN[24], RETR_CMD[24], CHOISE[24], CLO_TM[24], PGNO1[24], PRESS1[24], PGNO2[24], PRESS2[24], SPOT_PARAMS[24]
STRUC SPOT_TYPE INT GUN, S_PAIR_SLCT PAIR, COMMAND RETR, INT CLO_TM, INT PGNO1, REAL PRESS1, INT PGNO2, REAL PRESS2

;==============================
; External declarations:
;==============================
EXT USERSPOT (S_COMMAND :IN, SPOT_TYPE :IN )

;==============================
; Variables:
;==============================
DECL SPOT_TYPE SDEFAULT={GUN 1,PAIR #FIRST,RETR #OPN,CLO_TM 0,PGNO1 1,PRESS1 0.0,PGNO2 0,PRESS2 0.0}
DECL SPOT_TYPE S_ACT
DECL INT S_ACT_DELAY
DECL BOOL S_READY
;ENDFOLD (SPOTTECH GLOBALS)
;FOLD USER GLOBALS
;*******************************************
;Make your modifications -ONLY- here
;*******************************************
;==================================
; Userdefined Types
;==================================

;==================================
; Userdefined Externals
;==================================

;==================================
; Userdefined Variables
;==================================

FRAME valueframe

;FOLD Sack Offset
DECL INT SackTypeOffSetX[6,16]; SackType,SackNo
SackTypeOffSetX[1,1]=0
SackTypeOffSetX[1,2]=0
SackTypeOffSetX[1,3]=0
SackTypeOffSetX[1,4]=0
SackTypeOffSetX[1,5]=0
SackTypeOffSetX[1,6]=0
SackTypeOffSetX[1,7]=0
SackTypeOffSetX[1,8]=0
SackTypeOffSetX[1,9]=0
SackTypeOffSetX[1,10]=0
SackTypeOffSetX[1,11]=0
SackTypeOffSetX[1,12]=0
SackTypeOffSetX[1,13]=0
SackTypeOffSetX[1,14]=0
SackTypeOffSetX[1,15]=0
SackTypeOffSetX[1,16]=0

SackTypeOffSetX[2,1]=0
SackTypeOffSetX[2,2]=0
SackTypeOffSetX[2,3]=0
SackTypeOffSetX[2,4]=0
SackTypeOffSetX[2,5]=0
SackTypeOffSetX[2,6]=0
SackTypeOffSetX[2,7]=0
SackTypeOffSetX[2,8]=0
SackTypeOffSetX[2,9]=0
SackTypeOffSetX[2,10]=0
SackTypeOffSetX[2,11]=0
SackTypeOffSetX[2,12]=0
SackTypeOffSetX[2,13]=0
SackTypeOffSetX[2,14]=0
SackTypeOffSetX[2,15]=0
SackTypeOffSetX[2,16]=0

SackTypeOffSetX[3,1]=0
SackTypeOffSetX[3,2]=0
SackTypeOffSetX[3,3]=0
SackTypeOffSetX[3,4]=0
SackTypeOffSetX[3,5]=0
SackTypeOffSetX[3,6]=0
SackTypeOffSetX[3,7]=30
SackTypeOffSetX[3,8]=0
SackTypeOffSetX[3,9]=0
SackTypeOffSetX[3,10]=0
SackTypeOffSetX[3,11]=0
SackTypeOffSetX[3,12]=0
SackTypeOffSetX[3,13]=50
SackTypeOffSetX[3,14]=50
SackTypeOffSetX[3,15]=40
SackTypeOffSetX[3,16]=10

SackTypeOffSetX[4,1]=0
SackTypeOffSetX[4,2]=0
SackTypeOffSetX[4,3]=0
SackTypeOffSetX[4,4]=0
SackTypeOffSetX[4,5]=0
SackTypeOffSetX[4,6]=0
SackTypeOffSetX[4,7]=0
SackTypeOffSetX[4,8]=0
SackTypeOffSetX[4,9]=0
SackTypeOffSetX[4,10]=0
SackTypeOffSetX[4,11]=0
SackTypeOffSetX[4,12]=0
SackTypeOffSetX[4,13]=0
SackTypeOffSetX[4,14]=0
SackTypeOffSetX[4,15]=0
SackTypeOffSetX[4,16]=0

SackTypeOffSetX[5,1]=0
SackTypeOffSetX[5,2]=0
SackTypeOffSetX[5,3]=0
SackTypeOffSetX[5,4]=0
SackTypeOffSetX[5,5]=0
SackTypeOffSetX[5,6]=0
SackTypeOffSetX[5,7]=0
SackTypeOffSetX[5,8]=0
SackTypeOffSetX[5,9]=0
SackTypeOffSetX[5,10]=0
SackTypeOffSetX[5,11]=0
SackTypeOffSetX[5,12]=0
SackTypeOffSetX[5,13]=0
SackTypeOffSetX[5,14]=0
SackTypeOffSetX[5,15]=0
SackTypeOffSetX[5,16]=0

SackTypeOffSetX[6,1]=70
SackTypeOffSetX[6,2]=70
SackTypeOffSetX[6,3]=-40
SackTypeOffSetX[6,4]=-40
SackTypeOffSetX[6,5]=0
SackTypeOffSetX[6,6]=-20
SackTypeOffSetX[6,7]=-20
SackTypeOffSetX[6,8]=-20
SackTypeOffSetX[6,9]=-70
SackTypeOffSetX[6,10]=20
SackTypeOffSetX[6,11]=-70
SackTypeOffSetX[6,12]=20
SackTypeOffSetX[6,13]=-20
SackTypeOffSetX[6,14]=50
SackTypeOffSetX[6,15]=0
SackTypeOffSetX[6,16]=0


DECL INT SackTypeOffSetY[6,16]; SackType,SackNo

SackTypeOffSetY[1,1]=0
SackTypeOffSetY[1,2]=0
SackTypeOffSetY[1,3]=0
SackTypeOffSetY[1,4]=0
SackTypeOffSetY[1,5]=0
SackTypeOffSetY[1,6]=0
SackTypeOffSetY[1,7]=0
SackTypeOffSetY[1,8]=0
SackTypeOffSetY[1,9]=0
SackTypeOffSetY[1,10]=0
SackTypeOffSetY[1,11]=0
SackTypeOffSetY[1,12]=0
SackTypeOffSetY[1,13]=0
SackTypeOffSetY[1,14]=0
SackTypeOffSetY[1,15]=0
SackTypeOffSetY[1,16]=0

SackTypeOffSetY[2,1]=0
SackTypeOffSetY[2,2]=0
SackTypeOffSetY[2,3]=0
SackTypeOffSetY[2,4]=0
SackTypeOffSetY[2,5]=0
SackTypeOffSetY[2,6]=0
SackTypeOffSetY[2,7]=0
SackTypeOffSetY[2,8]=0
SackTypeOffSetY[2,9]=0
SackTypeOffSetY[2,10]=0
SackTypeOffSetY[2,11]=0
SackTypeOffSetY[2,12]=0
SackTypeOffSetY[2,13]=0
SackTypeOffSetY[2,14]=0
SackTypeOffSetY[2,15]=0
SackTypeOffSetY[2,16]=0

SackTypeOffSetY[3,1]=0
SackTypeOffSetY[3,2]=0
SackTypeOffSetY[3,3]=0
SackTypeOffSetY[3,4]=0
SackTypeOffSetY[3,5]=0
SackTypeOffSetY[3,6]=0
SackTypeOffSetY[3,7]=0
SackTypeOffSetY[3,8]=0
SackTypeOffSetY[3,9]=0
SackTypeOffSetY[3,10]=0
SackTypeOffSetY[3,11]=0
SackTypeOffSetY[3,12]=0
SackTypeOffSetY[3,13]=0
SackTypeOffSetY[3,14]=0
SackTypeOffSetY[3,15]=0
SackTypeOffSetY[3,16]=0

SackTypeOffSetY[4,1]=0
SackTypeOffSetY[4,2]=0
SackTypeOffSetY[4,3]=0
SackTypeOffSetY[4,4]=0
SackTypeOffSetY[4,5]=0
SackTypeOffSetY[4,6]=0
SackTypeOffSetY[4,7]=0
SackTypeOffSetY[4,8]=0
SackTypeOffSetY[4,9]=0
SackTypeOffSetY[4,10]=0
SackTypeOffSetY[4,11]=0
SackTypeOffSetY[4,12]=0
SackTypeOffSetY[4,13]=0
SackTypeOffSetY[4,14]=0
SackTypeOffSetY[4,15]=0
SackTypeOffSetY[4,16]=0

SackTypeOffSetY[5,1]=0
SackTypeOffSetY[5,2]=0
SackTypeOffSetY[5,3]=0
SackTypeOffSetY[5,4]=0
SackTypeOffSetY[5,5]=0
SackTypeOffSetY[5,6]=0
SackTypeOffSetY[5,7]=0
SackTypeOffSetY[5,8]=0
SackTypeOffSetY[5,9]=0
SackTypeOffSetY[5,10]=0
SackTypeOffSetY[5,11]=0
SackTypeOffSetY[5,12]=0
SackTypeOffSetY[5,13]=0
SackTypeOffSetY[5,14]=0
SackTypeOffSetY[5,15]=0
SackTypeOffSetY[5,16]=0

SackTypeOffSetY[6,1]=-100
SackTypeOffSetY[6,2]=-80
SackTypeOffSetY[6,3]=-130
SackTypeOffSetY[6,4]=-80
SackTypeOffSetY[6,5]=0
SackTypeOffSetY[6,6]=0
SackTypeOffSetY[6,7]=0
SackTypeOffSetY[6,8]=0
SackTypeOffSetY[6,9]=-40
SackTypeOffSetY[6,10]=-40
SackTypeOffSetY[6,11]=0
SackTypeOffSetY[6,12]=-20
SackTypeOffSetY[6,13]=0
SackTypeOffSetY[6,14]=0
SackTypeOffSetY[6,15]=0
SackTypeOffSetY[6,16]=0


;DECL INT 4SackTypeOffSetY[6,16]; SackType,SackNo

DECL INT OffsetX_4[2,8]
;Left
OffsetX_4[1,1]=0
OffsetX_4[1,2]=0
OffsetX_4[1,3]=0
OffsetX_4[1,4]=0
OffsetX_4[1,5]=0
OffsetX_4[1,6]=0
OffsetX_4[1,7]=0
OffsetX_4[1,8]=0
;Right
OffsetX_4[2,1]=0
OffsetX_4[2,2]=0
OffsetX_4[2,3]=0
OffsetX_4[2,4]=0
OffsetX_4[2,5]=0
OffsetX_4[2,6]=0
OffsetX_4[2,7]=0
OffsetX_4[2,8]=0

DECL INT OffsetY_4[2,8]
;Left
OffsetY_4[1,1]=0
OffsetY_4[1,2]=0
OffsetY_4[1,3]=0
OffsetY_4[1,4]=0
OffsetY_4[1,5]=0
OffsetY_4[1,6]=0
OffsetY_4[1,7]=0
OffsetY_4[1,8]=0
;Right
OffsetY_4[2,1]=0
OffsetY_4[2,2]=0
OffsetY_4[2,3]=0
OffsetY_4[2,4]=0
OffsetY_4[2,5]=0
OffsetY_4[2,6]=0
OffsetY_4[2,7]=0
OffsetY_4[2,8]=0

;ENDFOLD
DECL INT lifth=1
DECL INT rightn=2
DECL INT SackNoOffSet
DECL INT HIGHT6=50
DECL INT INT_NoPalLef
DECL INT INT_PLCRobSpd
DECL INT INT_NoPalRgh

DECL INT Debug=0

SIGNAL NoPalLef $IN[201] TO $IN[208];26  ;PLC Byte + 1
SIGNAL PLCRobSpd $IN[209] TO $IN[216];27
SIGNAL NoPalRgh $IN[217] TO $IN[224];28


SIGNAL EopSckNoLft $OUT[89] TO $OUT[96]
SIGNAL EopSckNoRgh $OUT[105] TO $OUT[112]
SIGNAL MonRunTim $OUT[113] TO $OUT[128]

;DECL INT INT_BagLinLef
;DECL INT INT_BagLinRgh
;SIGNAL BagLinLef $OUT[81] TO $IN[88];11  ;PLC Byte + 1
;SIGNAL BagLinRgh $OUT[97] TO $IN[104];13  ;PLC Byte + 1


;ENDFOLD (USER GLOBALS)
ENDDAT
